Staubli VAL3: unSelectItem.pgx

public program unSelectItem()
  local InstrItem l_sEvent
  local num i
  local num l_nSize
begin
  // deselect all
  call getSizeItem(l_nSize)
  for i=0 to (l_nSize-1)
    call getItem(l_sEvent,i)
    if find(l_sEvent.sType,"#")!=-1
      l_sEvent.sType=right(l_sEvent.sType,len(l_sEvent.sType)-1)
      call setItem(l_sEvent,i)
    endIf
  endFor
end
